FUNCTION_BLOCK FB_Module_Base
VAR_INPUT
	IC		: BOOL;
	Execute	: BOOL;
	Ack		: BOOL;
END_VAR

VAR_OUTPUT
	Ready		: BOOL;
	Failure		: BOOL;
	Done		: BOOL;
END_VAR

VAR
	tm		: S_Timeouts;
END_VAR

END_FUNCTION_BLOCK

(* stored: Version 1.1.0.1, ProductVersion 3.1.4024.11
   POU FB_Module_Base: Id {3a301875-b2bb-427d-a6fa-5afb38800442}, SpecialFunc None *)
